FUNCTION_BLOCK logiBUS_LED_strip_QXA (* Composite FB for LED strip output data *)
  (* Standard: 61499-2; Description: Copyright (c) 2026 HR Agrartechnik GmbH This program and the accompanying materials are made available under the terms of the Eclipse Public License 2.0 which is available at https://www.eclipse.org/legal/epl-2.0/ SPDX-License-Identifier: EPL-2.0 *)
  (* Version 1.0, 2026-02-23, Franz Höpfinger, HR Agrartechnik GmbH *)
  PACKAGE logiBUS::io::DO_LED;
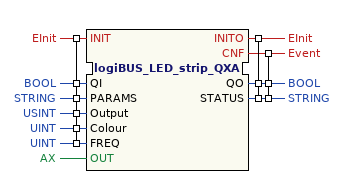
  EVENT_INPUT
    INIT : EInit WITH QI, PARAMS, Output, Colour, FREQ; (* Service Initialization *)
  END_EVENT
  EVENT_OUTPUT
    INITO : EInit WITH QO, STATUS; (* Initialization Confirm *)
    CNF WITH QO, STATUS; (* Confirmation of Requested Service *)
  END_EVENT
  VAR_INPUT
    QI : BOOL; (* Event Input Qualifier *)
    PARAMS : STRING; (* Service Parameters *)
    Output : USINT := LED_strip::Output_strip; (* Identify the Output Number of Strip *)
    Colour : UINT := LED_COLOURS::LED_GREEN; (* This identify the Colour. *)
    FREQ : UINT := LED_FREQ::LED_OFF; (* Define the LED Frequency and Priority *)
  END_VAR
  VAR_OUTPUT
    QO : BOOL; (* Event Output Qualifier *)
    STATUS : STRING; (* Service Status *)
  END_VAR
  SOCKETS
    OUT : adapter::types::unidirectional::AX; (* Output data to resource *)
  END_SOCKETS
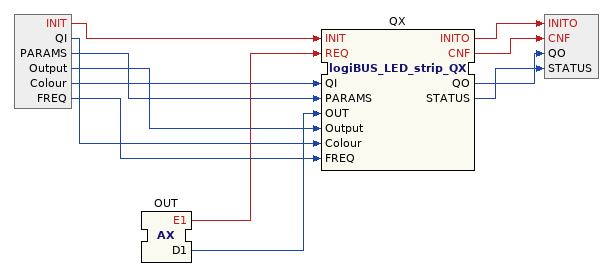
  FBS
    QX : logiBUS::io::DO_LED::logiBUS_LED_strip_QX;
  END_FBS
  EVENT_CONNECTIONS
    INIT TO QX.INIT;
    QX.INITO TO INITO;
    OUT.E1 TO QX.REQ;
    QX.CNF TO CNF;
  END_CONNECTIONS
  DATA_CONNECTIONS
    OUT.D1 TO QX.OUT;
    QI TO QX.QI;
    PARAMS TO QX.PARAMS;
    QX.QO TO QO;
    QX.STATUS TO STATUS;
    Output TO QX.Output;
    Colour TO QX.Colour;
    FREQ TO QX.FREQ;
  END_CONNECTIONS
END_FUNCTION_BLOCK
